Staubli VAL3: load.pgx

public program load(string x_sItem, num& x_nResult[])
  local string l_sPath
  local string l_sName
  local string l_sType
  local progItem l_pNull
  local string l_sMessage
begin
  // check the libPath
  call getType(l_sType)
  // load it
  if find(saveProg:libPath(),saveData:sPathProg)==-1
    x_nResult=saveProg:libLoad(saveData:sPathProg+l_sType)
    delay(0)
    if saveData:bDebug
      ? "loading PROG..."+saveData:sPathProg+l_sType
    endIf
  endIf
  // reload the edit template
  if isDefined(saveProg:pProg[x_sItem].sID) and x_sItem!=""
    // refresh the iD...
    saveProg:pProg[x_sItem].sID=x_sItem
    // update the select item
    pEdit=saveProg:pProg[x_sItem]
  elseIf x_sItem!=""
    // not FOUND
    call language:message(l_sMessage,-7)
    x_nResult=-1
    popUpMsg(l_sMessage+x_sItem)
    // use an empty one
    pEdit.sID=""
  endIf
end
